FUNCTION_BLOCK FB_TankController IMPLEMENTS I_TankController

VAR_IN_OUT
	nNum : INT;
END_VAR
VAR
END_VAR

{warning 'add method implementation '}
METHOD ApplyCooling
END_METHOD

{warning 'add method implementation '}
METHOD CheckSafety
END_METHOD

END_FUNCTION_BLOCK

(* stored: Version 1.1.0.1, ProductVersion 3.1.4024.16
   POU FB_TankController: Id {c5e85192-36f8-483e-b1a4-1c5b3e658233}, SpecialFunc None
   Method ApplyCooling: Id {426552bd-63fa-4d79-8c07-4fdfe2acc75d}
   Method CheckSafety: Id {8b875647-f6f6-45de-ab91-5423d7d1628d} *)
